Fanuc KAREL source: kt00240.KL

-- PROVISIONAL review KL for V1013-1; original PC SHA256 da6b56526cea41df86765dba95fd7b5ea72b4a5ed7dbff544c429b2cda165ece
-- Incomplete behavior may be omitted. Consult companion uncertainty JSON. Do not deploy.
PROGRAM KT00240
%NOLOCKGROUP
VAR
  I1 : INTEGER
  OUT : INTEGER
-- UNRESOLVED_DECL H2 type=002017
BEGIN
  -- UNRESOLVED_PC offsets 5-16; opcodes 2E,23
  -- UNRESOLVED_PC offsets 21-35; opcodes 2E,22,9D,33,B4
  -- UNRESOLVED_PC offsets 40-62; opcodes 21,22,9D,33,B3,47,23
  -- UNRESOLVED_PC offsets 67-71; opcodes 7F
END KT00240
